FUNCTION_BLOCK FB_TapButton
VAR_INPUT
END_VAR
VAR_OUTPUT
END_VAR
VAR
END_VAR

END_FUNCTION_BLOCK

(* stored: Version 1.1.0.1, ProductVersion 3.1.4024.12
   POU FB_TapButton: Id {0b04fee2-8e62-40ea-8cee-6a7f03323788}, SpecialFunc None *)
